// TIA Portal V17 export
// export: Created 2023-03-06T02:05:24.2289887Z, ExportSetting WithDefaults, DisplayName Totally Integrated Automation Portal, DisplayVersion V17 Update 4, DisplayName TIA Portal Openness, DisplayVersion V17 Update 4, DisplayName TIA Portal Version Control Interface, DisplayVersion V17, DisplayName STEP 7 Professional, DisplayVersion V17 Update 4, DisplayName STEP 7 Safety, DisplayVersion V17, DisplayName WinCC Professional, DisplayVersion V17 Update 4
ORGANIZATION_BLOCK "ProfiNet 10ms"   // OB30, LAD, CyclicInterrupt
{ S7_Optimized_Access := 'TRUE' }
VERSION : 0.1
// stored: AutoNumber true, IsIECCheckEnabled false, SetENOAutomatically false
   VAR_INPUT
      Initial_Call : Bool;   // Initial call of this OB
      Event_Count : Int;   // Events discarded
   END_VAR
   VAR_TEMP
      Ret_val : Int;
   END_VAR
BEGIN

REGION Network 1: Diagnostic Profinet Module (CPU is Module 1)
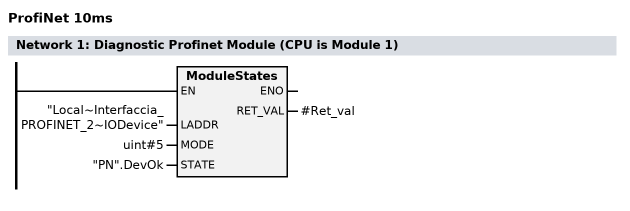
   RUNG wire#powerrail
      ModuleStates(LADDR := "Local~Interfaccia_PROFINET_2~IODevice", MODE := uint#5, STATE := "PN".DevOk, Ret_Val => #Ret_val)
   END_RUNG
   // the same network as SCL:
   #Ret_val := ModuleStates(LADDR := "Local~Interfaccia_PROFINET_2~IODevice",
                           MODE := uint#5,
                           STATE := "PN".DevOk);
END_REGION
END_ORGANIZATION_BLOCK
